FUNCTION_BLOCK FB_2Out IMPLEMENTS  I_ConveyerSection
VAR_INPUT
END_VAR
VAR_OUTPUT
END_VAR
VAR
	stRack	: ST_2Out;
	nStep	: UINT;
	bStart	: BOOL;
	_mDwnStrmHndShkIn	: BOOL;
	_mDwnStrmHndShkOut	: BOOL;
	_mUpStrmHndShkIn	: BOOL;
	_mUpStrmHndShkOut	: BOOL;
	_mId				: UINT;
	_mHMI				: ARRAY[0..15] OF BOOL;
	_mPosition			: INT;
END_VAR

Sequence();


PROPERTY DwnStrmHndShkIn : BOOL
SET
_mDwnStrmHndShkIn := DwnStrmHndShkIn;
END_SET
END_PROPERTY


PROPERTY DwnStrmHndShkOut : BOOL
GET
DwnStrmHndShkOut := _mDwnStrmHndShkOut;
END_GET
END_PROPERTY

{warning 'add property implementation'}
PROPERTY HMI : ARRAY [0..15] OF BOOL
GET
_mHMI[0] := stRack.ST_Out1.Output1;
_mHMI[1] := stRack.ST_Out1.Output2;
_mHMI[2] := stRack.ST_Out1.Output3;
_mHMI[3] := stRack.ST_Out1.Output4;
_mHMI[4] := stRack.ST_Out1.Output5;
_mHMI[5] := stRack.ST_Out1.Output6;
_mHMI[6] := stRack.ST_Out1.Output7;
_mHMI[7] := stRack.ST_Out1.Output8;
_mHMI[8] := stRack.ST_Out2.Output1;
_mHMI[9] := stRack.ST_Out2.Output2;
_mHMI[10] := stRack.ST_Out2.Output3;
_mHMI[11] := stRack.ST_Out2.Output4;
_mHMI[12] := stRack.ST_Out2.Output5;
_mHMI[13] := stRack.ST_Out2.Output6;
_mHMI[14] := stRack.ST_Out2.Output7;
_mHMI[15] := stRack.ST_Out2.Output8;

HMI := _mHMI;
END_GET
END_PROPERTY


PROPERTY Id : UINT
GET
Id := _mId;
END_GET
SET
_mId := Id;
END_SET
END_PROPERTY

{warning 'add property implementation'}
PROPERTY Pos : INT
GET
Pos := _mPosition;
END_GET
SET
_mPosition := Pos;
END_SET
END_PROPERTY


METHOD  Sequence : BOOL
IF bStart THEN
CASE nStep OF
0:
	stRack.ST_Out1.Output1 := TRUE;
	stRack.ST_Out2.Output1 := FALSE;
	IF _mDwnStrmHndShkIn THEN
		_mDwnStrmHndShkOut := FALSE;
	END_IF
	IF _mUpStrmHndShkIn THEN
		_mUpStrmHndShkOut := TRUE;
	END_IF
	nStep:=1;
1:
	stRack.ST_Out1.Output3 := TRUE;
	stRack.ST_Out2.Output3 := FALSE;
	IF _mDwnStrmHndShkIn THEN
		_mDwnStrmHndShkOut := TRUE;
	END_IF
		IF _mUpStrmHndShkIn THEN
		_mUpStrmHndShkOut := FALSE;
	END_IF
	nStep := 2;
2:
	stRack.ST_Out1.Output5 := TRUE;
	stRack.ST_Out2.Output5 := FALSE;
	IF _mDwnStrmHndShkIn THEN
		_mDwnStrmHndShkOut := FALSE;
	END_IF
		IF _mUpStrmHndShkIn THEN
		_mUpStrmHndShkOut := TRUE;
	END_IF
	nStep:=3;
3:
	stRack.ST_Out1.Output7 := TRUE;
	stRack.ST_Out2.Output7 := FALSE;
	IF _mDwnStrmHndShkIn THEN
		_mDwnStrmHndShkOut := TRUE;
	END_IF
		IF _mUpStrmHndShkIn THEN
		_mUpStrmHndShkOut := FALSE;
	END_IF
	nStep:=4;
4:
	stRack.ST_Out1.Output2 := TRUE;
	stRack.ST_Out2.Output2 := FALSE;
	IF _mDwnStrmHndShkIn THEN
		_mDwnStrmHndShkOut := FALSE;
	END_IF
		IF _mUpStrmHndShkIn THEN
		_mUpStrmHndShkOut := TRUE;
	END_IF
	nStep:=5;
5:
	stRack.ST_Out1.Output4 := TRUE;
	stRack.ST_Out2.Output4 := FALSE;
	IF _mDwnStrmHndShkIn THEN
		_mDwnStrmHndShkOut := TRUE;
	END_IF
		IF _mUpStrmHndShkIn THEN
		_mUpStrmHndShkOut := FALSE;
	END_IF
	nStep:=6;
6:
	stRack.ST_Out1.Output6 := TRUE;
	stRack.ST_Out2.Output6 := FALSE;
	IF _mDwnStrmHndShkIn THEN
		_mDwnStrmHndShkOut := FALSE;
	END_IF
		IF _mUpStrmHndShkIn THEN
		_mUpStrmHndShkOut := TRUE;
	END_IF
	nStep:=7;
7:
	stRack.ST_Out1.Output8 := TRUE;
	stRack.ST_Out2.Output8 := FALSE;
	IF _mDwnStrmHndShkIn THEN
		_mDwnStrmHndShkOut := TRUE;
	END_IF
		IF _mUpStrmHndShkIn THEN
		_mUpStrmHndShkOut := FALSE;
	END_IF
	nStep:=8;
8:
	stRack.ST_Out1.Output1 := FALSE;
	stRack.ST_Out2.Output1 := TRUE;
	IF _mDwnStrmHndShkIn THEN
		_mDwnStrmHndShkOut := FALSE;
	END_IF
		IF _mUpStrmHndShkIn THEN
		_mUpStrmHndShkOut := TRUE;
	END_IF
	nStep:=9;
9:
	stRack.ST_Out1.Output3 := FALSE;
	stRack.ST_Out2.Output3 := TRUE;
	IF _mDwnStrmHndShkIn THEN
		_mDwnStrmHndShkOut := TRUE;
	END_IF
		IF _mUpStrmHndShkIn THEN
		_mUpStrmHndShkOut := FALSE;
	END_IF
	nStep:=10;
10:
	stRack.ST_Out1.Output5 := FALSE;
	stRack.ST_Out2.Output5 := TRUE;
	IF _mDwnStrmHndShkIn THEN
		_mDwnStrmHndShkOut := FALSE;
	END_IF
		IF _mUpStrmHndShkIn THEN
		_mUpStrmHndShkOut := TRUE;
	END_IF
	nStep:=11;
11:
	stRack.ST_Out1.Output7 := FALSE;
	stRack.ST_Out2.Output7 := TRUE;
	IF _mDwnStrmHndShkIn THEN
		_mDwnStrmHndShkOut := TRUE;
	END_IF
		IF _mUpStrmHndShkIn THEN
		_mUpStrmHndShkOut := FALSE;
	END_IF
	nStep:=12;
12:
	stRack.ST_Out1.Output2 := FALSE;
	stRack.ST_Out2.Output2 := TRUE;
	IF _mDwnStrmHndShkIn THEN
		_mDwnStrmHndShkOut := FALSE;
	END_IF
		IF _mUpStrmHndShkIn THEN
		_mUpStrmHndShkOut := TRUE;
	END_IF
	nStep:=13;
13:
	stRack.ST_Out1.Output4 := FALSE;
	stRack.ST_Out2.Output4 := TRUE;
	IF _mDwnStrmHndShkIn THEN
		_mDwnStrmHndShkOut := TRUE;
	END_IF
	nStep:=14;
14:
	stRack.ST_Out1.Output6 := FALSE;
	stRack.ST_Out2.Output6 := TRUE;
	IF _mDwnStrmHndShkIn THEN
		_mDwnStrmHndShkOut := FALSE;
	END_IF
		IF _mUpStrmHndShkIn THEN
		_mUpStrmHndShkOut := FALSE;
	END_IF
	nStep:=15;
15:
	stRack.ST_Out1.Output8 := FALSE;
	stRack.ST_Out2.Output8 := TRUE;
	IF _mDwnStrmHndShkIn THEN
		_mDwnStrmHndShkOut := TRUE;
	END_IF
		IF _mUpStrmHndShkIn THEN
		_mUpStrmHndShkOut := FALSE;
	END_IF
	nStep:=0;

END_CASE
END_IF

THIS^._mDwnStrmHndShkOut := THIS^._mUpStrmHndShkIn;
END_METHOD


METHOD startSequence : BOOL
bStart := TRUE;
nStep := 0;
stRack.ST_Out1.Output1 := FALSE;
stRack.ST_Out1.Output2 := FALSE;
stRack.ST_Out1.Output3 := FALSE;
stRack.ST_Out1.Output4 := FALSE;
stRack.ST_Out1.Output5 := FALSE;
stRack.ST_Out1.Output6 := FALSE;
stRack.ST_Out1.Output7 := FALSE;
stRack.ST_Out1.Output8 := FALSE;
stRack.ST_Out2.Output1 := FALSE;
stRack.ST_Out2.Output2 := FALSE;
stRack.ST_Out2.Output3 := FALSE;
stRack.ST_Out2.Output4 := FALSE;
stRack.ST_Out2.Output5 := FALSE;
stRack.ST_Out2.Output6 := FALSE;
stRack.ST_Out2.Output7 := FALSE;
stRack.ST_Out2.Output8 := FALSE;
END_METHOD

METHOD stopSequence : BOOL
bStart := FALSE;
nStep :=0;
THIS^._mDwnStrmHndShkOut := FALSE;
THIS^._mUpStrmHndShkOut := FALSE;
END_METHOD


PROPERTY UpStrmHndShkIn : BOOL
SET
_mUpStrmHndShkIn := UpStrmHndShkIn;
END_SET
END_PROPERTY


PROPERTY UpStrmHndShkOut : BOOL
GET
UpStrmHndShkOut	:= _mUpStrmHndShkOut;
END_GET
END_PROPERTY

END_FUNCTION_BLOCK

(* stored: Version 1.1.0.1, ProductVersion 3.1.4024.6
   POU FB_2Out: Id {8f0b6be3-790d-4526-b456-e791a7000168}, SpecialFunc None
   Property DwnStrmHndShkIn: Id {db8b557a-bf99-4314-b18c-55865b9e3807}
   Set Set: Id {46bb6fac-d546-4ebb-89e7-0bc0230631a3}
   Property DwnStrmHndShkOut: Id {e8325890-966b-45e3-b328-0a830ac6c858}
   Get Get: Id {7ca479e2-6fa7-4119-8b61-af5ca1c27042}
   Property HMI: Id {88b1e012-a4f6-4a38-a194-adf4c9f428ff}
   Get Get: Id {ee557eae-8270-425e-be0c-ff4de02cd022}
   Property Id: Id {bc8254dd-500e-4ed6-871e-3c6ca3334b6f}
   Get Get: Id {49179a91-2cce-438c-a953-60549b6ae108}
   Set Set: Id {2a19f696-4bc9-4674-a05d-c469eef0d24c}
   Property Pos: Id {36880dc7-5032-48de-a69e-59b180a445fc}
   Get Get: Id {5ac75453-7f88-4dc5-9a14-d2f808c21729}
   Set Set: Id {42181b56-a11e-4c0e-911a-e87bde2c9303}
   Method Sequence: Id {26a65c71-9c29-4aaf-ab06-63f349f40e97}
   Method startSequence: Id {7d1d1a32-46fb-4152-b149-03a30baf4eda}
   Method stopSequence: Id {a9e97247-44f4-4dd1-b3d2-4eea92d2a7c8}
   Property UpStrmHndShkIn: Id {c90ddcc8-a3de-499d-8686-35fc4fb39c71}
   Set Set: Id {ed93e6d8-9b76-42c1-b11d-99e96e1bfbbe}
   Property UpStrmHndShkOut: Id {a3608a1f-a166-4725-8e92-d1cbf89d83e5}
   Get Get: Id {6d53efc2-586e-4718-a9e2-bf8ed8e557f8} *)
